Staubli VAL3: remGetTCPVals.pgx

program remGetTCPVals(string& sReturn[] (dimensions=1))
  local trsf trTCP
begin
  // Return the Cartesian values of the TCP
  //
  logMsg("call remSetIPVals")
  trTCP=tSensorTool.trsf
  sReturn="GETTCPVALS"
  sReturn=sReturn+" "+toString(sNumConv,trTCP.x)
  sReturn=sReturn+" "+toString(sNumConv,trTCP.y)
  sReturn=sReturn+" "+toString(sNumConv,trTCP.z)
  sReturn=sReturn+" "+toString(sNumConv,trTCP.rx)
  sReturn=sReturn+" "+toString(sNumConv,trTCP.ry)
  sReturn=sReturn+" "+toString(sNumConv,trTCP.rz)
end
